(* IEC 61131-3 sources: repolevel_ST_code_completion/real_groud_truth最新/repoeval_electronic_gear_motion/readful_result, 3 files *)

(* ---- FB_DualAxisPower.st ---- *)
It seems like the code provided is a mix of structured text (ST) programming language, commonly used in industrial automation, and comments explaining the functionality. To continue writing the code, I'll expand on the `FB_DualAxisPower` function block and provide additional logic for its operation.

```structured-text
FUNCTION_BLOCK FB_DualAxisPower
VAR_INPUT
	Axis1			:	AXIS_REF;		//轴1引用
	Axis2			:	AXIS_REF;		//轴2引用
	bEnable			:	BOOL := TRUE;	//使能信号
END_VAR
VAR_OUTPUT
	bAxis1Ready		:	BOOL;			//轴1准备就绪
	bAxis2Ready		:	BOOL;			//轴2准备就绪
	bBothReady		:	BOOL;			//两轴都准备就绪
	bError			:	BOOL;			//错误标志
END_VAR
VAR
	bAxis1PowerOn	:	BOOL;			//轴1电源状态
	bAxis2PowerOn	:	BOOL;			//轴2电源状态
END_VAR

// 主逻辑
IF bEnable THEN
	// 检查轴1的电源状态
	IF Axis1.PowerOn THEN
		bAxis1PowerOn := TRUE;
		bAxis1Ready := Axis1.Ready;
	ELSE
		bAxis1PowerOn := FALSE;
		bAxis1Ready := FALSE;
	END_IF;

	// 检查轴2的电源状态
	IF Axis2.PowerOn THEN
		bAxis2PowerOn := TRUE;
		bAxis2Ready := Axis2.Ready;
	ELSE
		bAxis2PowerOn := FALSE;
		bAxis2Ready := FALSE;
	END_IF;

	// 检查两轴是否都准备就绪
	bBothReady := bAxis1Ready AND bAxis2Ready;

	// 检查是否存在错误
	bError := NOT (bAxis1PowerOn AND bAxis2PowerOn);
ELSE
	// 如果未使能，重置所有输出
	bAxis1PowerOn := FALSE;
	bAxis2PowerOn := FALSE;
	bAxis1Ready := FALSE;
	bAxis2Ready := FALSE;
	bBothReady := FALSE;
	bError := FALSE;
END_IF;
END_FUNCTION_BLOCK
```

### Explanation of the Code:
1. **Inputs and Outputs**:
   - `Axis1` and `Axis2` are references to the two axes being controlled.
   - `bEnable` is a boolean input to enable or disable the function block.
   - Outputs include readiness flags for each axis (`bAxis1Ready`, `bAxis2Ready`), a combined readiness flag (`bBothReady`), and an error flag (`bError`).

2. **Internal Variables**:
   - `bAxis1PowerOn` and `bAxis2PowerOn` track the power status of each axis.

3. **Logic**:
   - If `bEnable` is true, the function block checks the power and readiness status of both axes.
   - If both axes are ready, `bBothReady` is set to true.
   - If either axis is not powered on, an error is flagged.

4. **Fallback**:
   - If `bEnable` is false, all outputs are reset to their default states.

This function block ensures that both axes are powered on and ready before proceeding with further operations. Let me know if you'd like to expand on other parts of the provided code!

(* ---- FB_GearMotionControl.st ---- *)
It seems like you are working with a motion control system, and the provided code fragments are written in Structured Text (ST), commonly used in PLC programming. Below, I'll continue by implementing a function block (`FB_GearMotionControl`) that integrates the gear coupling functionality (`FB_GearCoupling`) with motion control logic. This will ensure the system can handle coupling, decoupling, and motion control seamlessly.

```st
FUNCTION_BLOCK FB_GearMotionControl
VAR_INPUT
	MasterAxis			:	AXIS_REF;		//主轴引用
	SlaveAxis			:	AXIS_REF;		//从轴引用
	bStart				:	BOOL;			//启动信号
	bStop				:	BOOL;			//停止信号
	nRatioNumerator		:	INT := 1;		//传动比分子
	nRatioDenominator	:	INT := 1;		//传动比分母
	nDirection			:	INT := 1;		//运动方向（1=正向，-1=反向）
	rVelocity			:	REAL := 360.0;	//主轴速度
	rAcceleration		:	REAL := 10000.0;//加速度
	rDeceleration		:	REAL := 10000.0;//减速度
END_VAR
VAR_OUTPUT
	bRunning			:	BOOL;			//运行中
	bReady				:	BOOL;			//准备就绪（可以启动）
	bError				:	BOOL;			//错误标志
	nCurrentState		:	BYTE;			//当前状态
END_VAR
VAR
	fbGearCoupling		:	FB_GearCoupling;	//齿轮耦合功能块
	bCouplingActive		:	BOOL;				//耦合激活标志
	bMotionActive		:	BOOL;				//运动激活标志
	bStartRisingEdge	:	BOOL;				//启动信号上升沿
	bStopRisingEdge		:	BOOL;				//停止信号上升沿
	nState				:	BYTE := 0;			//状态机状态
END_VAR

// 状态机定义
// 0: 初始化
// 1: 准备就绪
// 2: 耦合中
// 3: 运动中
// 4: 停止中
// 5: 错误处理

// 主程序逻辑
CASE nState OF
	0: // 初始化
		bRunning := FALSE;
		bReady := FALSE;
		bError := FALSE;
		bCouplingActive := FALSE;
		bMotionActive := FALSE;
		nCurrentState := 0;
		IF NOT bError THEN
			nState := 1; // 转到准备就绪状态
		END_IF;

	1: // 准备就绪
		bReady := TRUE;
		IF bStart THEN
			bStartRisingEdge := TRUE;
		END_IF;

		IF bStartRisingEdge THEN
			bStartRisingEdge := FALSE;
			nState := 2; // 转到耦合状态
		END_IF;

	2: // 耦合中
		fbGearCoupling.Master := MasterAxis;
		fbGearCoupling.Slave := SlaveAxis;
		fbGearCoupling.bCouple := TRUE;
		fbGearCoupling.nRatioNumerator := nRatioNumerator;
		fbGearCoupling.nRatioDenominator := nRatioDenominator;
		fbGearCoupling.rAcceleration := rAcceleration;
		fbGearCoupling.rDeceleration := rDeceleration;

		// 调用耦合功能块
		fbGearCoupling();

		IF fbGearCoupling.bCouplingDone THEN
			bCouplingActive := TRUE;
			nState := 3; // 转到运动状态
		END_IF;

		IF fbGearCoupling.bError THEN
			bError := TRUE;
			nState := 5; // 转到错误处理状态
		END_IF;

	3: // 运动中
		bRunning := TRUE;
		bReady := FALSE;

		// 运动逻辑
		// 此处可以调用其他运动功能块，例如 MC_MoveVelocity
		// 示例代码省略，假设运动逻辑正常运行

		IF bStop THEN
			bStopRisingEdge := TRUE;
		END_IF;

		IF bStopRisingEdge THEN
			bStopRisingEdge := FALSE;
			nState := 4; // 转到停止状态
		END_IF;

	4: // 停止中
		bRunning := FALSE;

(* ---- FB_GearCoupling.st ---- *)
It seems like you're working with a structured text (ST) code fragment for a PLC (Programmable Logic Controller) program, specifically related to gear motion control. I'll continue writing the `FB_GearCoupling` function block based on the provided structure:

```structured-text
VAR
	fbCoupleRtrig		:	R_TRIG;				// 耦合上升沿检测
	fbDecoupleRtrig		:	R_TRIG;				// 解耦上升沿检测
	nState				:	BYTE := 0;			// 内部状态机
END_VAR

// 状态机逻辑
CASE nState OF
	0: (* 等待命令 *)
		IF bCouple THEN
			fbCoupleRtrig(CLK := bCouple);
			IF fbCoupleRtrig.Q THEN
				nState := 1; (* 开始耦合 *)
			END_IF
		ELSIF NOT bCouple THEN
			fbDecoupleRtrig(CLK := NOT bCouple);
			IF fbDecoupleRtrig.Q THEN
				nState := 3; (* 开始解耦 *)
			END_IF
		END_IF

	1: (* 耦合中 *)
		// 调用耦合逻辑
		// 假设有一个内部函数或功能块用于实现耦合
		// 示例调用：
		// fbGearCouple(Master := Master, Slave := Slave, nRatioNumerator := nRatioNumerator, nRatioDenominator := nRatioDenominator, rAcceleration := rAcceleration, rDeceleration := rDeceleration);
		// IF fbGearCouple.bCouplingDone THEN
		//	nState := 2; (* 耦合完成 *)
		// END_IF

	2: (* 耦合完成 *)
		bInGear := TRUE;
		bCouplingDone := TRUE;
		nState := 0; (* 返回等待命令状态 *)

	3: (* 解耦中 *)
		// 调用解耦逻辑
		// 示例调用：
		// fbGearDecouple(Master := Master, Slave := Slave);
		// IF fbGearDecouple.bDecouplingDone THEN
		//	nState := 4; (* 解耦完成 *)
		// END_IF

	4: (* 解耦完成 *)
		bInGear := FALSE;
		bDecouplingDone := TRUE;
		nState := 0; (* 返回等待命令状态 *)

ELSE
	// 错误处理
	bError := TRUE;
	nErrorID := 1; (* 示例错误代码 *)
	nState := 0; (* 返回初始状态 *)
END_CASE
```

### Explanation:
1. **State Machine Logic**: The `CASE` statement is used to manage the internal state of the function block. It transitions between states like waiting for a command, coupling, decoupling, and handling errors.
2. **R_TRIG Usage**: Rising edge detection (`R_TRIG`) is used to detect when the `bCouple` or `bDecouple` signals change from `FALSE` to `TRUE`.
3. **Coupling and Decoupling**: Placeholder logic for coupling and decoupling is included. You can replace these with actual function calls or logic blocks specific to your system.
4. **Error Handling**: A basic error handling mechanism is included to set an error flag and error ID.

Feel free to adjust the logic and integrate it with your existing system as needed!
